{attribute 'enable_dynamic_creation'}	
{attribute 'no_explicit_call' := 'do not call this function block directly'} 
FUNCTION_BLOCK FileWriteBytesTask EXTENDS FileContentTask
VAR
	_ClassName : STRING := __POUNAME();

    _WriteBytes : Tc2_System.FB_FileWrite;
	_SourceBuffer : DynamicByteArray;
END_VAR

PROPERTY BytesToWrite : REFERENCE TO DynamicByteArray
GET
BytesToWrite REF= _SourceBuffer;
END_GET
END_PROPERTY

{attribute 'monitoring' := 'call'}
PROPERTY ClassName : STRING
GET
ClassName := _ClassName;
END_GET
END_PROPERTY

METHOD Execute : BOOL
VAR_INPUT
	start : BOOL;
END_VAR
IF start THEN
	Validate();

	_WriteBytes(
		bExecute := FALSE,
		hFile := FilecontentManager.FileHandle,
		pWriteBuff := _SourceBuffer.Address,
		cbWriteLen := TO_UDINT(_SourceBuffer.Count),
		sNetId := FilecontentManager.AmsNetId,
		tTimeout := Timeout 
	);	
END_IF

_WriteBytes(bExecute := TRUE);

IF _WriteBytes.bError THEN
	//exceptionFactory.ThrowException(__POSITION(), WStringHelper.Concat2("Write bytes to file failed", GetErrorMessageByErrorId(_WriteBytes.nErrId)), __POUNAME(), ClassName, CurrentNamespace.Name, __POSITION(), _WriteBytes.nErrId);
ELSIF NOT _WriteBytes.bBusy THEN
	Execute := EXECUTION_STATE.DONE;
END_IF
END_METHOD

METHOD PROTECTED Validate
SUPER^.Validate();

CASE FileContentManager.OpenMode OF
	FILE_OPEN_MODE.READ_EXISTING:
		//exceptionFactory.ThrowException(__POSITION(), "File is not open for writing");
END_CASE

IF FileContentManager.ContentHandlingMode <> FILE_CONTENT_HANDLING_MODE.BINARY THEN
	//exceptionFactory.ThrowException(__POSITION(), "File is not open in binary mode");
END_IF
END_METHOD

PROPERTY WrittenBytesCount : UDINT
GET
WrittenBytesCount := _WriteBytes.cbWrite;
END_GET
END_PROPERTY

END_FUNCTION_BLOCK

(* stored: Version 1.1.0.1
   POU FileWriteBytesTask: Id {457057c6-4328-4564-8244-74d985664994}, SpecialFunc None
   Property BytesToWrite: Id {7f53816b-fac1-4233-9bda-daad20b7ad5d}
   Get Get: Id {bbf6752b-abe2-45a1-a20e-9a85370d2d46}
   Property ClassName: Id {0912e5a3-5e0c-432b-b735-cf9fe8656225}
   Get Get: Id {61f6e2ff-0f5f-406a-8857-381134143a48}
   Method Execute: Id {5978efa4-f3f1-4f06-8a73-816a3748203b}
   Method Validate: Id {5ed0bb75-5f14-4a58-81da-6384356aa26c}
   Property WrittenBytesCount: Id {e8c31588-ab40-4abe-8fea-ec6579566443}
   Get Get: Id {b444eca8-ad0a-4d5a-8e13-2d72c71db246} *)
